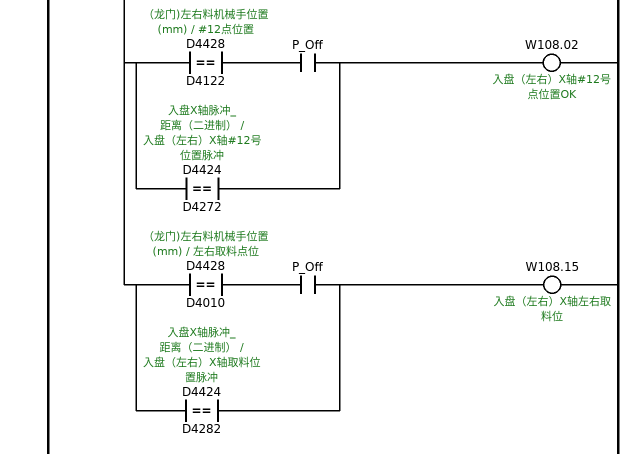
; [picture p264: 入盘机械 / 伺服参数设定, rungs 33-33]
; rung 33: 左右机械手所处位置 / 第一排12点
LD P_On
OUT TR0
LD=SL(303) D4428 D4100  ; （龙门)左右料机械手位置(mm), （龙门）左右#1号点位置
AND P_Off
OR=L(301) D4424 D4250  ; 入盘X轴脉冲_距离（二进制）, 入盘（左右）X轴#1号位置脉冲
ANDLD
OUT W107.07  ; 入盘（左右）X轴#1号点位置ok
LD TR0
LD=SL(303) D4428 D4102  ; （龙门)左右料机械手位置(mm), #2号点位置
AND P_Off
OR=L(301) D4424 D4252  ; 入盘X轴脉冲_距离（二进制）, 入盘（左右）X轴#2号位置脉冲
ANDLD
OUT W107.08  ; 入盘（左右）X轴#2号点位置OK
LD TR0
LD=SL(303) D4428 D4104  ; （龙门)左右料机械手位置(mm), #3点位置
AND P_Off
OR=L(301) D4424 D4254  ; 入盘X轴脉冲_距离（二进制）, 入盘（左右）X轴#3号位置脉冲)
ANDLD
OUT W107.09  ; 入盘（左右）X轴#3号点位置OK
LD TR0
LD=SL(303) D4428 D4106  ; （龙门)左右料机械手位置(mm), #4点位置
AND P_Off
OR=L(301) D4424 D4256  ; 入盘X轴脉冲_距离（二进制）, 入盘（左右）X轴#4号位置脉冲
ANDLD
OUT W107.10  ; 入盘（左右）X轴#4号点位置OK
LD TR0
LD=SL(303) D4428 D4108  ; （龙门)左右料机械手位置(mm), #5点位置
AND P_Off
OR=L(301) D4424 D4258  ; 入盘X轴脉冲_距离（二进制）, 入盘（左右）X轴#5号位置脉冲
ANDLD
OUT W107.11  ; 入盘（左右）X轴#5号点位置OK
LD TR0
LD=SL(303) D4428 D4110  ; （龙门)左右料机械手位置(mm), #6点位置
AND P_Off
OR=L(301) D4424 D4260  ; 入盘X轴脉冲_距离（二进制）, 入盘（左右）X轴#6号位置脉冲
ANDLD
OUT W107.12  ; 入盘（左右）X轴#6号点位置OK
LD TR0
LD=SL(303) D4428 D4112  ; （龙门)左右料机械手位置(mm), #7点位置
AND P_Off
OR=L(301) D4424 D4262  ; 入盘X轴脉冲_距离（二进制）, 入盘（左右）X轴#7号位置脉冲
ANDLD
OUT W107.13  ; 入盘（左右）X轴#7号点位置OK
LD TR0
LD=SL(303) D4428 D4114  ; （龙门)左右料机械手位置(mm), #8点位置
AND P_Off
OR=L(301) D4424 D4264  ; 入盘X轴脉冲_距离（二进制）, 入盘（左右）X轴#8号位置脉冲
ANDLD
OUT W107.14  ; 入盘（左右）X轴#8号点位置OK
LD TR0
LD=SL(303) D4428 D4116  ; （龙门)左右料机械手位置(mm), #9点位置
AND P_Off
OR=L(301) D4424 D4266  ; 入盘X轴脉冲_距离（二进制）, 入盘（左右）X轴#9号位置脉冲
ANDLD
OUT W107.15  ; 入盘（左右）X轴#9号点位置OK
LD TR0
LD=SL(303) D4428 D4118  ; （龙门)左右料机械手位置(mm), #10点位置
AND P_Off
OR=L(301) D4424 D4268  ; 入盘X轴脉冲_距离（二进制）, 入盘（左右）X轴#10号位置脉冲
ANDLD
OUT W108.00  ; 入盘（左右）X轴#10号点位置OK
LD TR0
LD=SL(303) D4428 D4120  ; （龙门)左右料机械手位置(mm), #11点位置
AND P_Off
OR=L(301) D4424 D4270  ; 入盘X轴脉冲_距离（二进制）, 入盘（左右）X轴#11号位置脉冲
ANDLD
OUT W108.01  ; 入盘（左右）X轴#11号点位置OK
LD TR0
LD=SL(303) D4428 D4122  ; （龙门)左右料机械手位置(mm), #12点位置
AND P_Off
OR=L(301) D4424 D4272  ; 入盘X轴脉冲_距离（二进制）, 入盘（左右）X轴#12号位置脉冲
ANDLD
OUT W108.02  ; 入盘（左右）X轴#12号点位置OK
LD TR0
LD=SL(303) D4428 D4010  ; （龙门)左右料机械手位置(mm), 左右取料点位
AND P_Off
OR=L(301) D4424 D4282  ; 入盘X轴脉冲_距离（二进制）, 入盘（左右）X轴取料位置脉冲
ANDLD
OUT W108.15  ; 入盘（左右）X轴左右取料位

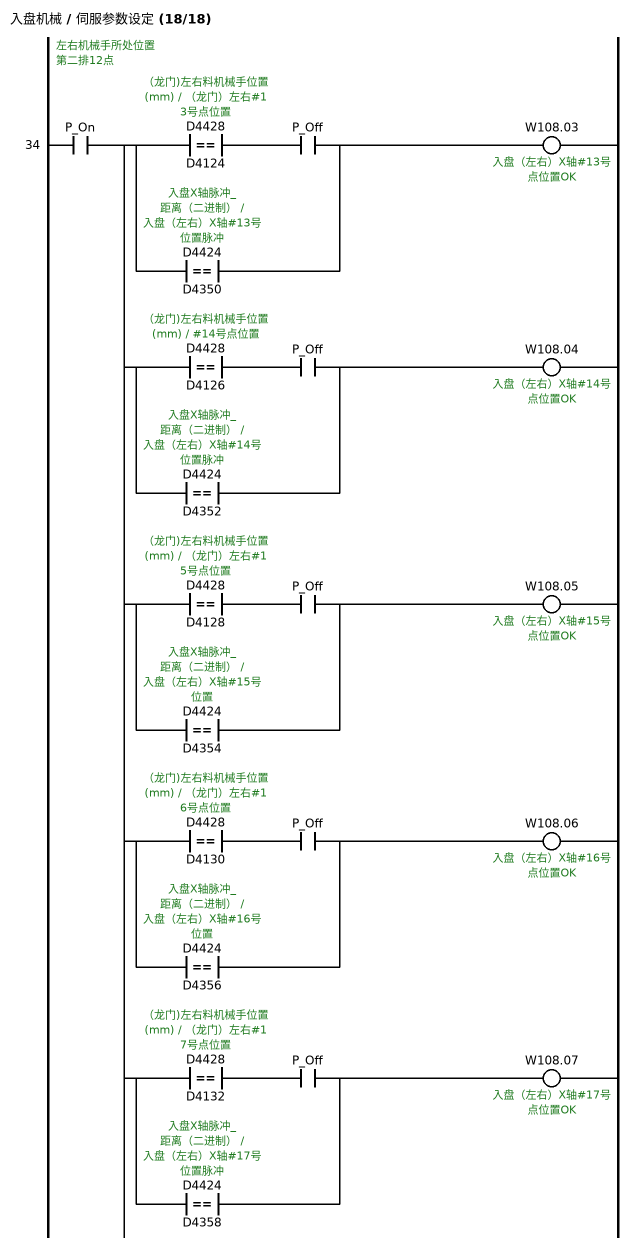

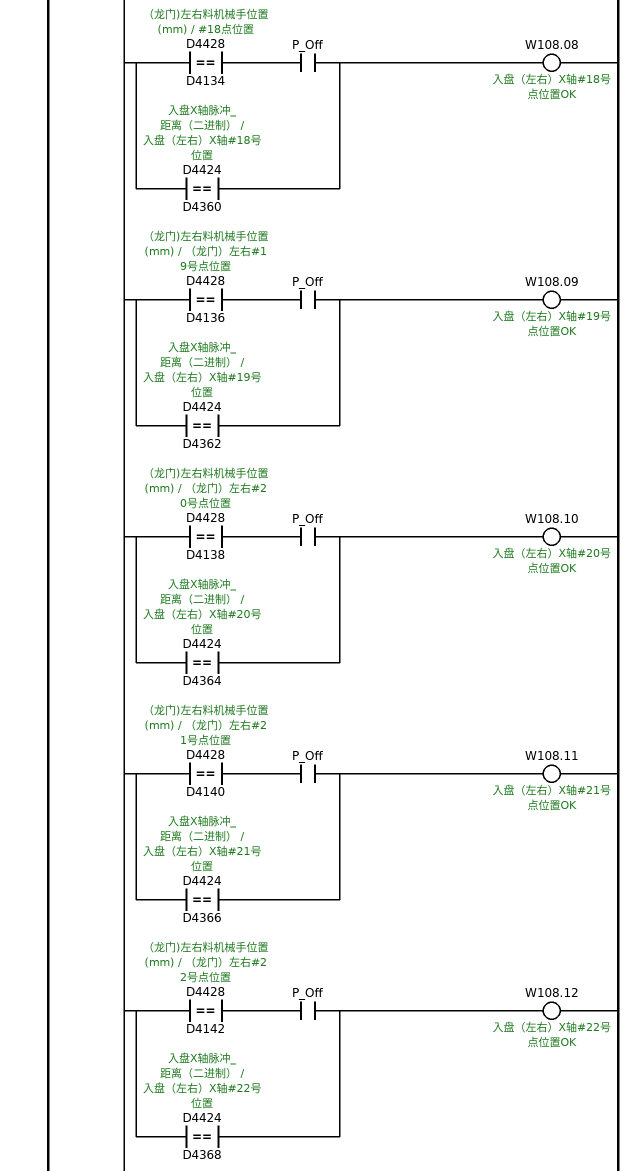

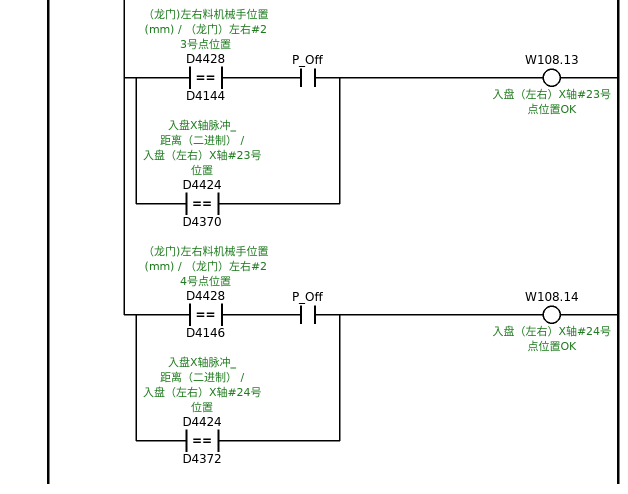
; rung 34: 左右机械手所处位置 / 第二排12点
LD P_On
OUT TR0
LD=SL(303) D4428 D4124  ; （龙门)左右料机械手位置(mm), （龙门）左右#13号点位置
AND P_Off
OR=L(301) D4424 D4350  ; 入盘X轴脉冲_距离（二进制）, 入盘（左右）X轴#13号位置脉冲
ANDLD
OUT W108.03  ; 入盘（左右）X轴#13号点位置OK
LD TR0
LD=SL(303) D4428 D4126  ; （龙门)左右料机械手位置(mm), #14号点位置
AND P_Off
OR=L(301) D4424 D4352  ; 入盘X轴脉冲_距离（二进制）, 入盘（左右）X轴#14号位置脉冲
ANDLD
OUT W108.04  ; 入盘（左右）X轴#14号点位置OK
LD TR0
LD=SL(303) D4428 D4128  ; （龙门)左右料机械手位置(mm), （龙门）左右#15号点位置
AND P_Off
OR=L(301) D4424 D4354  ; 入盘X轴脉冲_距离（二进制）, 入盘（左右）X轴#15号位置
ANDLD
OUT W108.05  ; 入盘（左右）X轴#15号点位置OK
LD TR0
LD=SL(303) D4428 D4130  ; （龙门)左右料机械手位置(mm), （龙门）左右#16号点位置
AND P_Off
OR=L(301) D4424 D4356  ; 入盘X轴脉冲_距离（二进制）, 入盘（左右）X轴#16号位置
ANDLD
OUT W108.06  ; 入盘（左右）X轴#16号点位置OK
LD TR0
LD=SL(303) D4428 D4132  ; （龙门)左右料机械手位置(mm), （龙门）左右#17号点位置
AND P_Off
OR=L(301) D4424 D4358  ; 入盘X轴脉冲_距离（二进制）, 入盘（左右）X轴#17号位置脉冲
ANDLD
OUT W108.07  ; 入盘（左右）X轴#17号点位置OK
LD TR0
LD=SL(303) D4428 D4134  ; （龙门)左右料机械手位置(mm), #18点位置
AND P_Off
OR=L(301) D4424 D4360  ; 入盘X轴脉冲_距离（二进制）, 入盘（左右）X轴#18号位置
ANDLD
OUT W108.08  ; 入盘（左右）X轴#18号点位置OK
LD TR0
LD=SL(303) D4428 D4136  ; （龙门)左右料机械手位置(mm), （龙门）左右#19号点位置
AND P_Off
OR=L(301) D4424 D4362  ; 入盘X轴脉冲_距离（二进制）, 入盘（左右）X轴#19号位置
ANDLD
OUT W108.09  ; 入盘（左右）X轴#19号点位置OK
LD TR0
LD=SL(303) D4428 D4138  ; （龙门)左右料机械手位置(mm), （龙门）左右#20号点位置
AND P_Off
OR=L(301) D4424 D4364  ; 入盘X轴脉冲_距离（二进制）, 入盘（左右）X轴#20号位置
ANDLD
OUT W108.10  ; 入盘（左右）X轴#20号点位置OK
LD TR0
LD=SL(303) D4428 D4140  ; （龙门)左右料机械手位置(mm), （龙门）左右#21号点位置
AND P_Off
OR=L(301) D4424 D4366  ; 入盘X轴脉冲_距离（二进制）, 入盘（左右）X轴#21号位置
ANDLD
OUT W108.11  ; 入盘（左右）X轴#21号点位置OK
LD TR0
LD=SL(303) D4428 D4142  ; （龙门)左右料机械手位置(mm), （龙门）左右#22号点位置
AND P_Off
OR=L(301) D4424 D4368  ; 入盘X轴脉冲_距离（二进制）, 入盘（左右）X轴#22号位置
ANDLD
OUT W108.12  ; 入盘（左右）X轴#22号点位置OK
LD TR0
LD=SL(303) D4428 D4144  ; （龙门)左右料机械手位置(mm), （龙门）左右#23号点位置
AND P_Off
OR=L(301) D4424 D4370  ; 入盘X轴脉冲_距离（二进制）, 入盘（左右）X轴#23号位置
ANDLD
OUT W108.13  ; 入盘（左右）X轴#23号点位置OK
LD TR0
LD=SL(303) D4428 D4146  ; （龙门)左右料机械手位置(mm), （龙门）左右#24号点位置
AND P_Off
OR=L(301) D4424 D4372  ; 入盘X轴脉冲_距离（二进制）, 入盘（左右）X轴#24号位置
ANDLD
OUT W108.14  ; 入盘（左右）X轴#24号点位置OK

### Section 外部输出及轴控运动

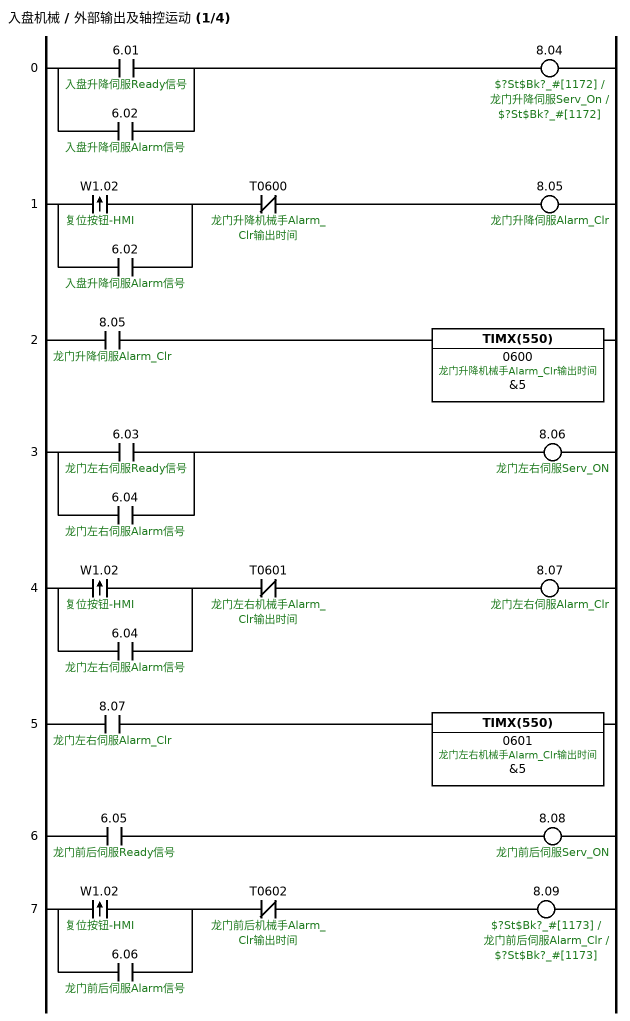
; rung 0
LD 6.01  ; 入盘升降伺服Ready信号
OR 6.02  ; 入盘升降伺服Alarm信号
OUT 8.04  ; $?St$Bk?_#[1172] / 龙门升降伺服Serv_On / $?St$Bk?_#[1172]
; rung 1
@LD W1.02  ; 复位按钮-HMI
OR 6.02  ; 入盘升降伺服Alarm信号
ANDNOT T0600  ; 龙门升降机械手Alarm_Clr输出时间
OUT 8.05  ; 龙门升降伺服Alarm_Clr
; rung 2
LD 8.05  ; 龙门升降伺服Alarm_Clr
TIMX(550) 0600 &5  ; 龙门升降机械手Alarm_Clr输出时间
; rung 3
LD 6.03  ; 龙门左右伺服Ready信号
OR 6.04  ; 龙门左右伺服Alarm信号
OUT 8.06  ; 龙门左右伺服Serv_ON
; rung 4
@LD W1.02  ; 复位按钮-HMI
OR 6.04  ; 龙门左右伺服Alarm信号
ANDNOT T0601  ; 龙门左右机械手Alarm_Clr输出时间
OUT 8.07  ; 龙门左右伺服Alarm_Clr
; rung 5
LD 8.07  ; 龙门左右伺服Alarm_Clr
TIMX(550) 0601 &5  ; 龙门左右机械手Alarm_Clr输出时间
; rung 6
LD 6.05  ; 龙门前后伺服Ready信号
OUT 8.08  ; 龙门前后伺服Serv_ON
; rung 7
@LD W1.02  ; 复位按钮-HMI
OR 6.06  ; 龙门前后伺服Alarm信号
ANDNOT T0602  ; 龙门前后机械手Alarm_Clr输出时间
OUT 8.09  ; $?St$Bk?_#[1173] / 龙门前后伺服Alarm_Clr / $?St$Bk?_#[1173]

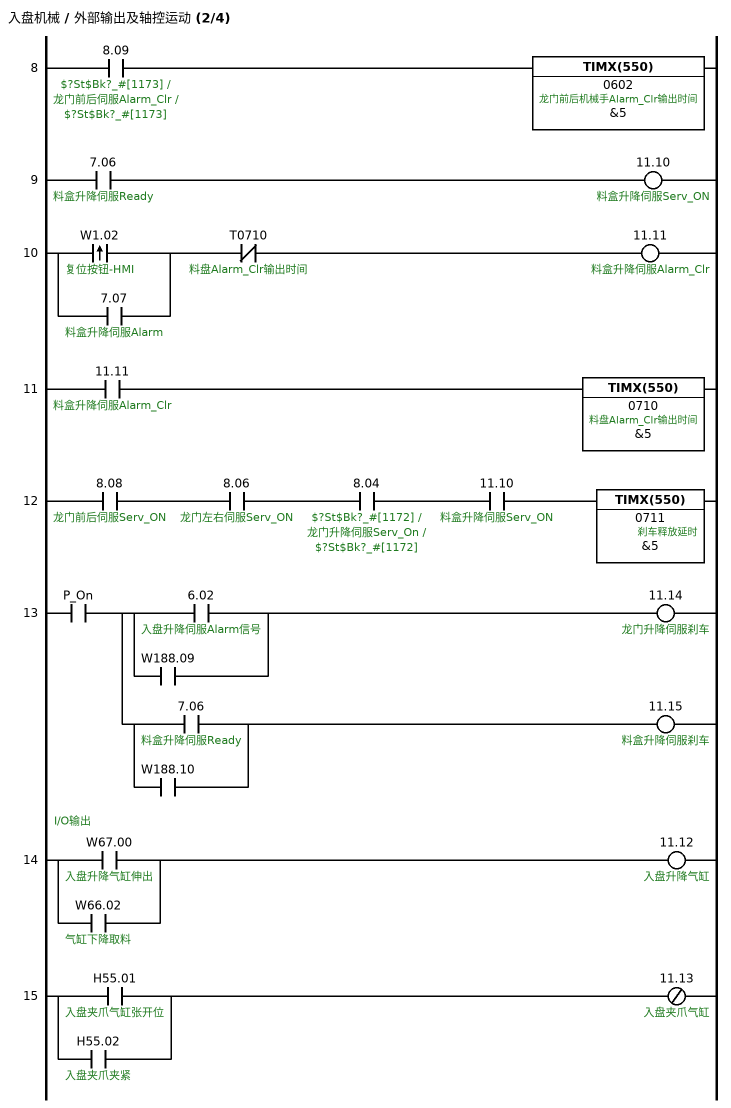
; rung 8
LD 8.09  ; $?St$Bk?_#[1173] / 龙门前后伺服Alarm_Clr / $?St$Bk?_#[1173]
TIMX(550) 0602 &5  ; 龙门前后机械手Alarm_Clr输出时间
; rung 9
LD 7.06  ; 料盒升降伺服Ready
OUT 11.10  ; 料盒升降伺服Serv_ON
; rung 10
@LD W1.02  ; 复位按钮-HMI
OR 7.07  ; 料盒升降伺服Alarm
ANDNOT T0710  ; 料盘Alarm_Clr输出时间
OUT 11.11  ; 料盒升降伺服Alarm_Clr
; rung 11
LD 11.11  ; 料盒升降伺服Alarm_Clr
TIMX(550) 0710 &5  ; 料盘Alarm_Clr输出时间
; rung 12
LD 8.08  ; 龙门前后伺服Serv_ON
AND 8.06  ; 龙门左右伺服Serv_ON
AND 8.04  ; $?St$Bk?_#[1172] / 龙门升降伺服Serv_On / $?St$Bk?_#[1172]
AND 11.10  ; 料盒升降伺服Serv_ON
TIMX(550) 0711 &5  ; 刹车释放延时
; rung 13
LD P_On
OUT TR0
LD 6.02  ; 入盘升降伺服Alarm信号
OR W188.09
ANDLD
OUT 11.14  ; 龙门升降伺服刹车
LD TR0
LD 7.06  ; 料盒升降伺服Ready
OR W188.10
ANDLD
OUT 11.15  ; 料盒升降伺服刹车
; rung 14: I/O输出
LD W67.00  ; 入盘升降气缸伸出
OR W66.02  ; 气缸下降取料
OUT 11.12  ; 入盘升降气缸
; rung 15
LD H55.01  ; 入盘夹爪气缸张开位
OR H55.02  ; 入盘夹爪夹紧
OUTNOT 11.13  ; 入盘夹爪气缸

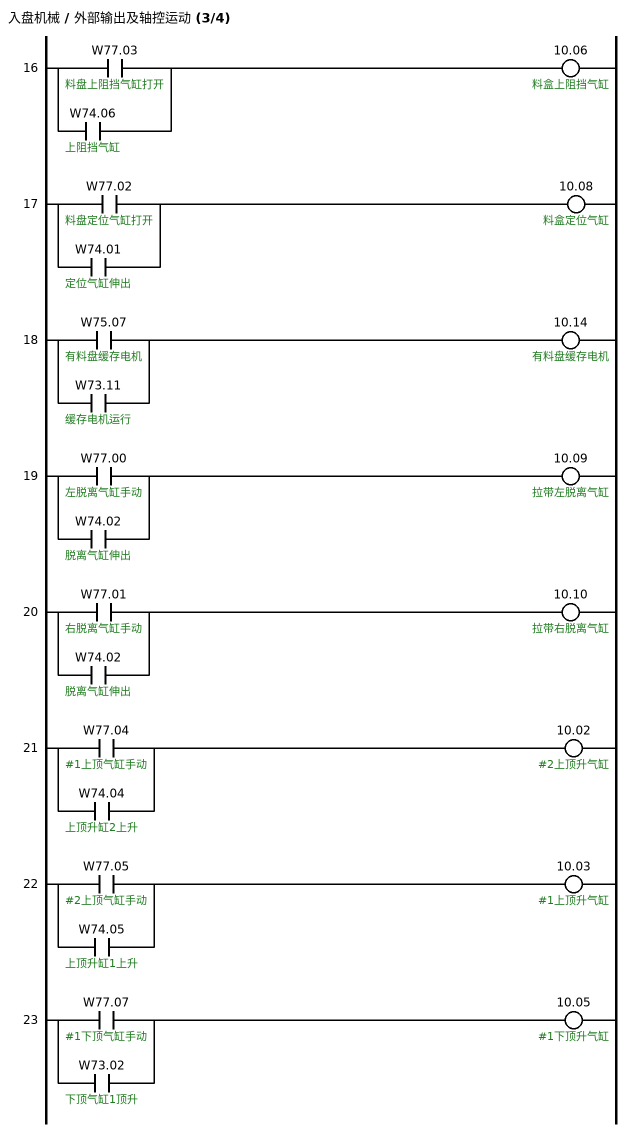
; rung 16
LD W77.03  ; 料盘上阻挡气缸打开
OR W74.06  ; 上阻挡气缸
OUT 10.06  ; 料盒上阻挡气缸
; rung 17
LD W77.02  ; 料盘定位气缸打开
OR W74.01  ; 定位气缸伸出
OUT 10.08  ; 料盒定位气缸
; rung 18
LD W75.07  ; 有料盘缓存电机
OR W73.11  ; 缓存电机运行
OUT 10.14  ; 有料盘缓存电机
; rung 19
LD W77.00  ; 左脱离气缸手动
OR W74.02  ; 脱离气缸伸出
OUT 10.09  ; 拉带左脱离气缸
; rung 20
LD W77.01  ; 右脱离气缸手动
OR W74.02  ; 脱离气缸伸出
OUT 10.10  ; 拉带右脱离气缸
; rung 21
LD W77.04  ; #1上顶气缸手动
OR W74.04  ; 上顶升缸2上升
OUT 10.02  ; #2上顶升气缸
; rung 22
LD W77.05  ; #2上顶气缸手动
OR W74.05  ; 上顶升缸1上升
OUT 10.03  ; #1上顶升气缸
; rung 23
LD W77.07  ; #1下顶气缸手动
OR W73.02  ; 下顶气缸1顶升
OUT 10.05  ; #1下顶升气缸

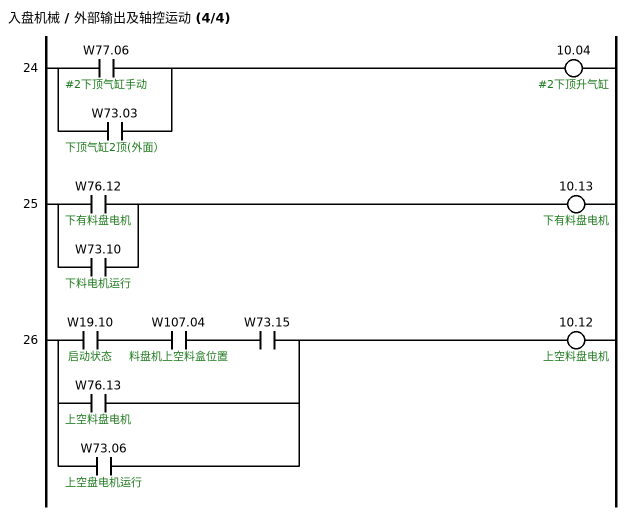
; rung 24
LD W77.06  ; #2下顶气缸手动
OR W73.03  ; 下顶气缸2顶(外面）
OUT 10.04  ; #2下顶升气缸
; rung 25
LD W76.12  ; 下有料盘电机
OR W73.10  ; 下料电机运行
OUT 10.13  ; 下有料盘电机
; rung 26
LD W19.10  ; 启动状态
AND W107.04  ; 料盘机上空料盒位置
AND W73.15
OR W76.13  ; 上空料盘电机
OR W73.06  ; 上空盘电机运行
OUT 10.12  ; 上空料盘电机

### Section 自动报警

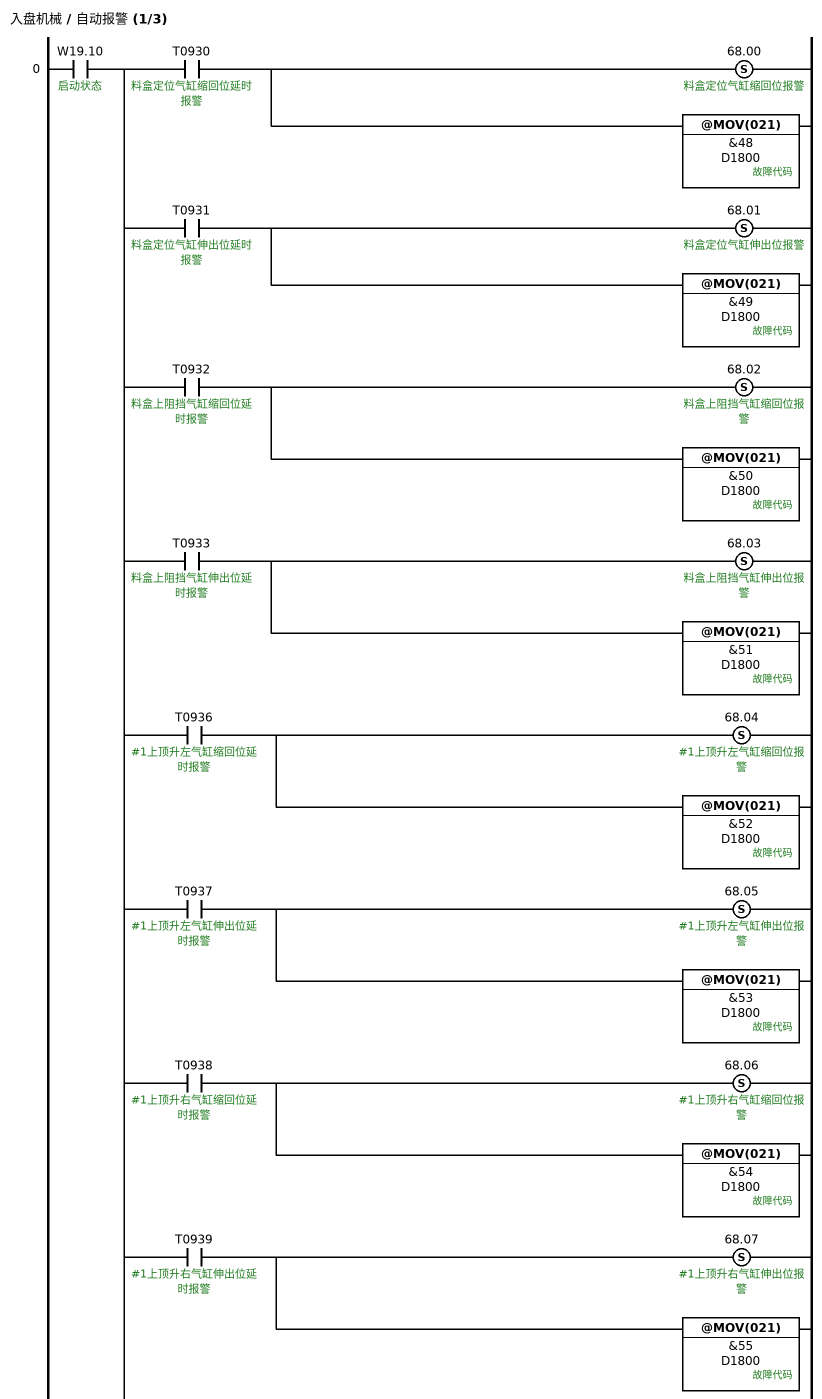

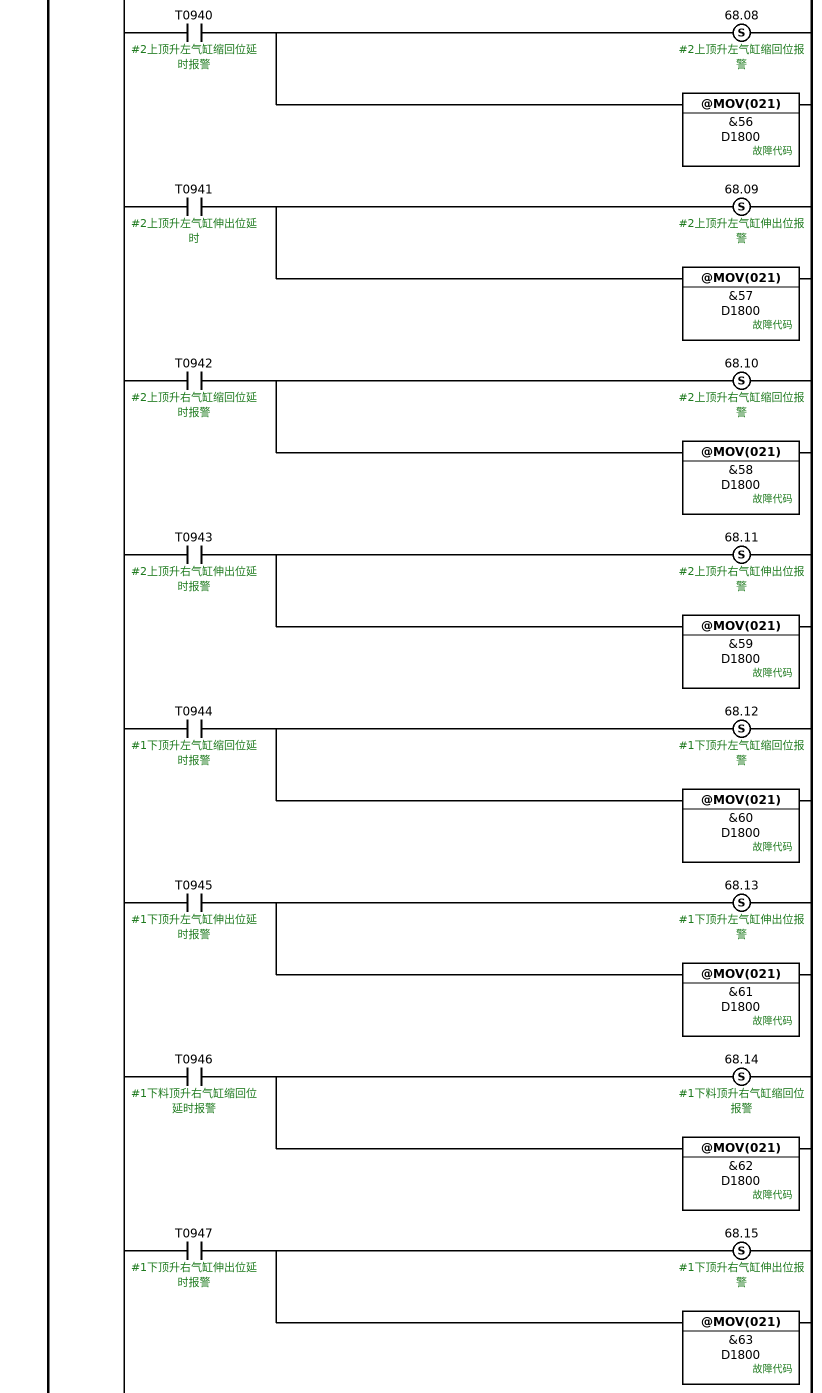

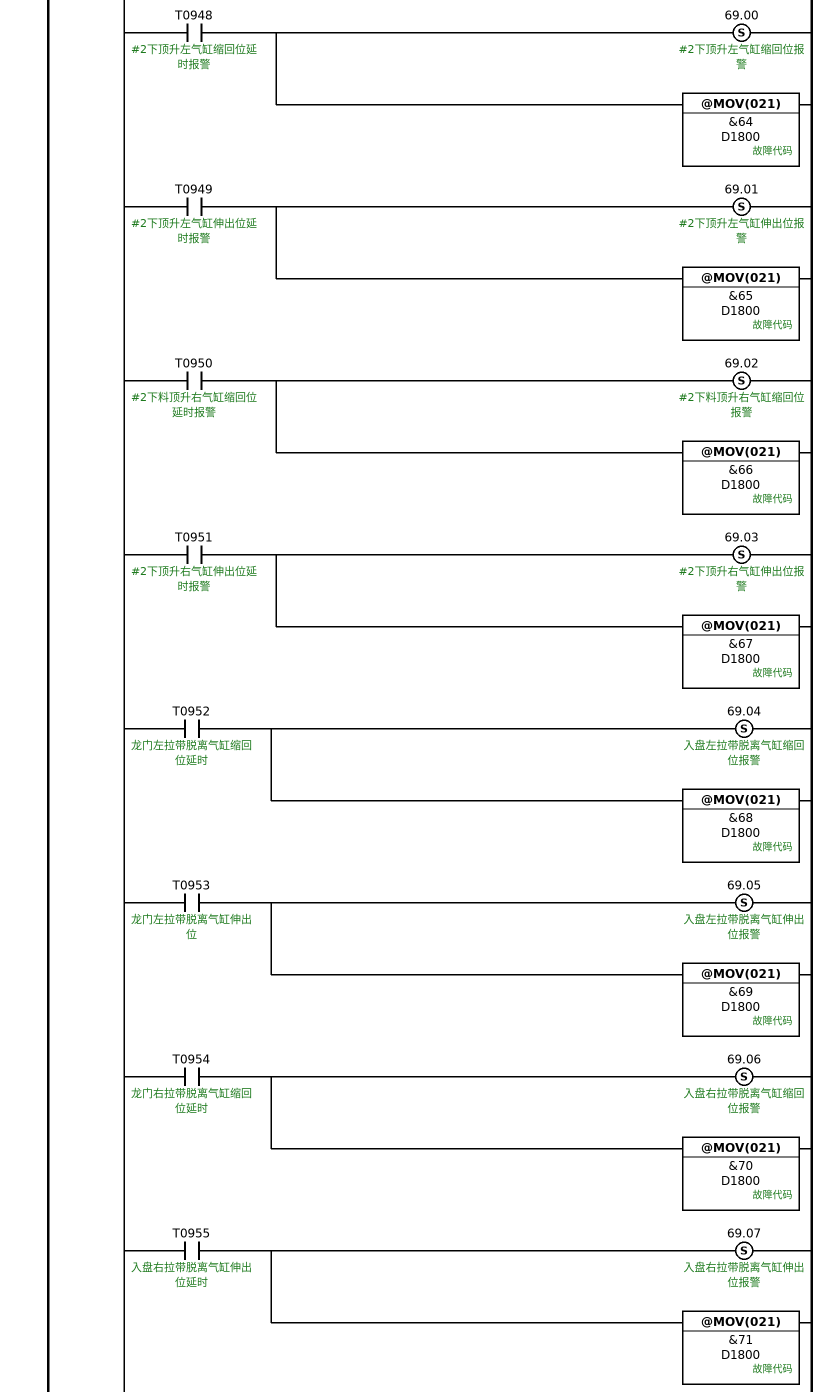

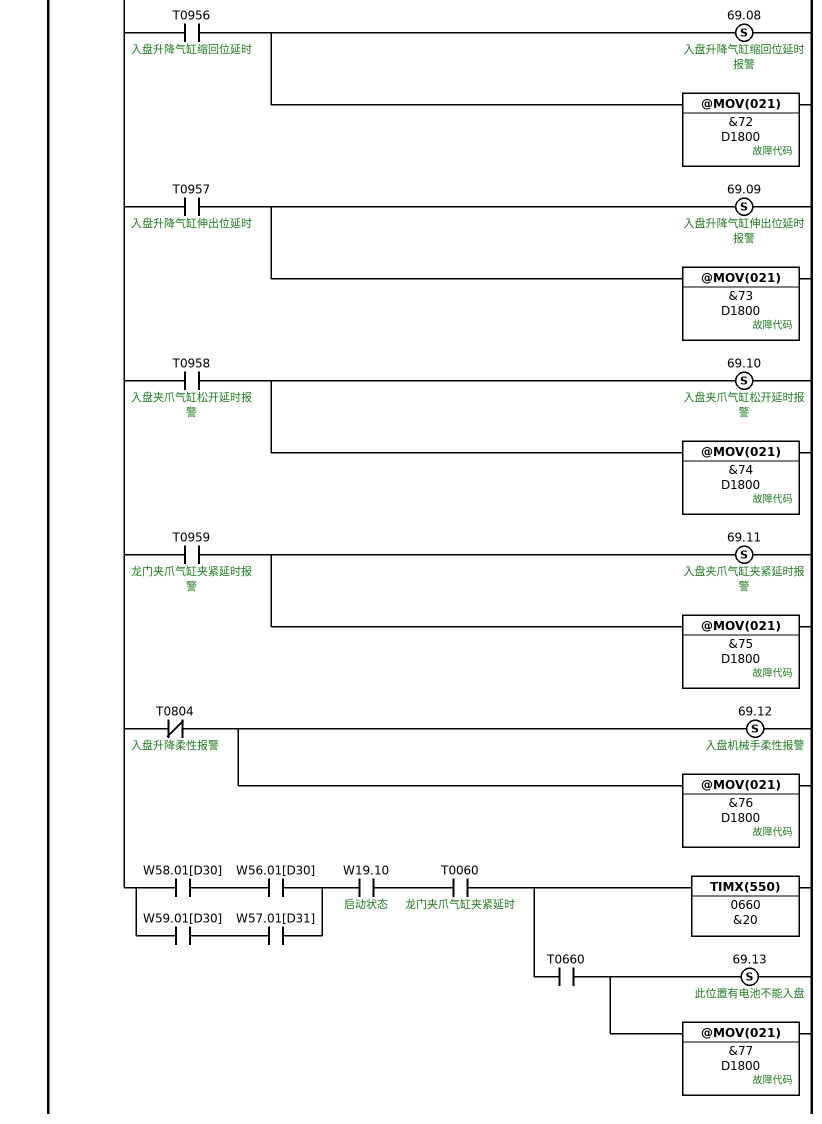
; rung 0
LD W19.10  ; 启动状态
OUT TR0
AND T0930  ; 料盒定位气缸缩回位延时报警
SET 68.00  ; 料盒定位气缸缩回位报警
@MOV(021) &48 D1800  ; 故障代码
LD TR0
AND T0931  ; 料盒定位气缸伸出位延时报警
SET 68.01  ; 料盒定位气缸伸出位报警
@MOV(021) &49 D1800  ; 故障代码
LD TR0
AND T0932  ; 料盒上阻挡气缸缩回位延时报警
SET 68.02  ; 料盒上阻挡气缸缩回位报警
@MOV(021) &50 D1800  ; 故障代码
LD TR0
AND T0933  ; 料盒上阻挡气缸伸出位延时报警
SET 68.03  ; 料盒上阻挡气缸伸出位报警
@MOV(021) &51 D1800  ; 故障代码
LD TR0
AND T0936  ; #1上顶升左气缸缩回位延时报警
SET 68.04  ; #1上顶升左气缸缩回位报警
@MOV(021) &52 D1800  ; 故障代码
LD TR0
AND T0937  ; #1上顶升左气缸伸出位延时报警
SET 68.05  ; #1上顶升左气缸伸出位报警
@MOV(021) &53 D1800  ; 故障代码
LD TR0
AND T0938  ; #1上顶升右气缸缩回位延时报警
SET 68.06  ; #1上顶升右气缸缩回位报警
@MOV(021) &54 D1800  ; 故障代码
LD TR0
AND T0939  ; #1上顶升右气缸伸出位延时报警
SET 68.07  ; #1上顶升右气缸伸出位报警
@MOV(021) &55 D1800  ; 故障代码
LD TR0
AND T0940  ; #2上顶升左气缸缩回位延时报警
SET 68.08  ; #2上顶升左气缸缩回位报警
@MOV(021) &56 D1800  ; 故障代码
LD TR0
AND T0941  ; #2上顶升左气缸伸出位延时
SET 68.09  ; #2上顶升左气缸伸出位报警
@MOV(021) &57 D1800  ; 故障代码
LD TR0
AND T0942  ; #2上顶升右气缸缩回位延时报警
SET 68.10  ; #2上顶升右气缸缩回位报警
@MOV(021) &58 D1800  ; 故障代码
LD TR0
AND T0943  ; #2上顶升右气缸伸出位延时报警
SET 68.11  ; #2上顶升右气缸伸出位报警
@MOV(021) &59 D1800  ; 故障代码
LD TR0
AND T0944  ; #1下顶升左气缸缩回位延时报警
SET 68.12  ; #1下顶升左气缸缩回位报警
@MOV(021) &60 D1800  ; 故障代码
LD TR0
AND T0945  ; #1下顶升左气缸伸出位延时报警
SET 68.13  ; #1下顶升左气缸伸出位报警
@MOV(021) &61 D1800  ; 故障代码
LD TR0
AND T0946  ; #1下料顶升右气缸缩回位延时报警
SET 68.14  ; #1下料顶升右气缸缩回位报警
@MOV(021) &62 D1800  ; 故障代码
LD TR0
AND T0947  ; #1下顶升右气缸伸出位延时报警
SET 68.15  ; #1下顶升右气缸伸出位报警
@MOV(021) &63 D1800  ; 故障代码
LD TR0
AND T0948  ; #2下顶升左气缸缩回位延时报警
SET 69.00  ; #2下顶升左气缸缩回位报警
@MOV(021) &64 D1800  ; 故障代码
LD TR0
AND T0949  ; #2下顶升左气缸伸出位延时报警
SET 69.01  ; #2下顶升左气缸伸出位报警
@MOV(021) &65 D1800  ; 故障代码
LD TR0
AND T0950  ; #2下料顶升右气缸缩回位延时报警
SET 69.02  ; #2下料顶升右气缸缩回位报警
@MOV(021) &66 D1800  ; 故障代码
LD TR0
AND T0951  ; #2下顶升右气缸伸出位延时报警
SET 69.03  ; #2下顶升右气缸伸出位报警
@MOV(021) &67 D1800  ; 故障代码
LD TR0
AND T0952  ; 龙门左拉带脱离气缸缩回位延时
SET 69.04  ; 入盘左拉带脱离气缸缩回位报警
@MOV(021) &68 D1800  ; 故障代码
LD TR0
AND T0953  ; 龙门左拉带脱离气缸伸出位
SET 69.05  ; 入盘左拉带脱离气缸伸出位报警
@MOV(021) &69 D1800  ; 故障代码
LD TR0
AND T0954  ; 龙门右拉带脱离气缸缩回位延时
SET 69.06  ; 入盘右拉带脱离气缸缩回位报警
@MOV(021) &70 D1800  ; 故障代码
LD TR0
AND T0955  ; 入盘右拉带脱离气缸伸出位延时
SET 69.07  ; 入盘右拉带脱离气缸伸出位报警
@MOV(021) &71 D1800  ; 故障代码
LD TR0
AND T0956  ; 入盘升降气缸缩回位延时
SET 69.08  ; 入盘升降气缸缩回位延时报警
@MOV(021) &72 D1800  ; 故障代码
LD TR0
AND T0957  ; 入盘升降气缸伸出位延时
SET 69.09  ; 入盘升降气缸伸出位延时报警
@MOV(021) &73 D1800  ; 故障代码
LD TR0
AND T0958  ; 入盘夹爪气缸松开延时报警
SET 69.10  ; 入盘夹爪气缸松开延时报警
@MOV(021) &74 D1800  ; 故障代码
LD TR0
AND T0959  ; 龙门夹爪气缸夹紧延时报警
SET 69.11  ; 入盘夹爪气缸夹紧延时报警
@MOV(021) &75 D1800  ; 故障代码
LD TR0
ANDNOT T0804  ; 入盘升降柔性报警
SET 69.12  ; 入盘机械手柔性报警
@MOV(021) &76 D1800  ; 故障代码
LD TR0
LD W58.01[D30]
AND W56.01[D30]
LD W59.01[D30]
AND W57.01[D31]
ORLD
ANDLD
AND W19.10  ; 启动状态
AND T0060  ; 龙门夹爪气缸夹紧延时
TIMX(550) 0660 &20
AND T0660
SET 69.13  ; 此位置有电池不能入盘
@MOV(021) &77 D1800  ; 故障代码

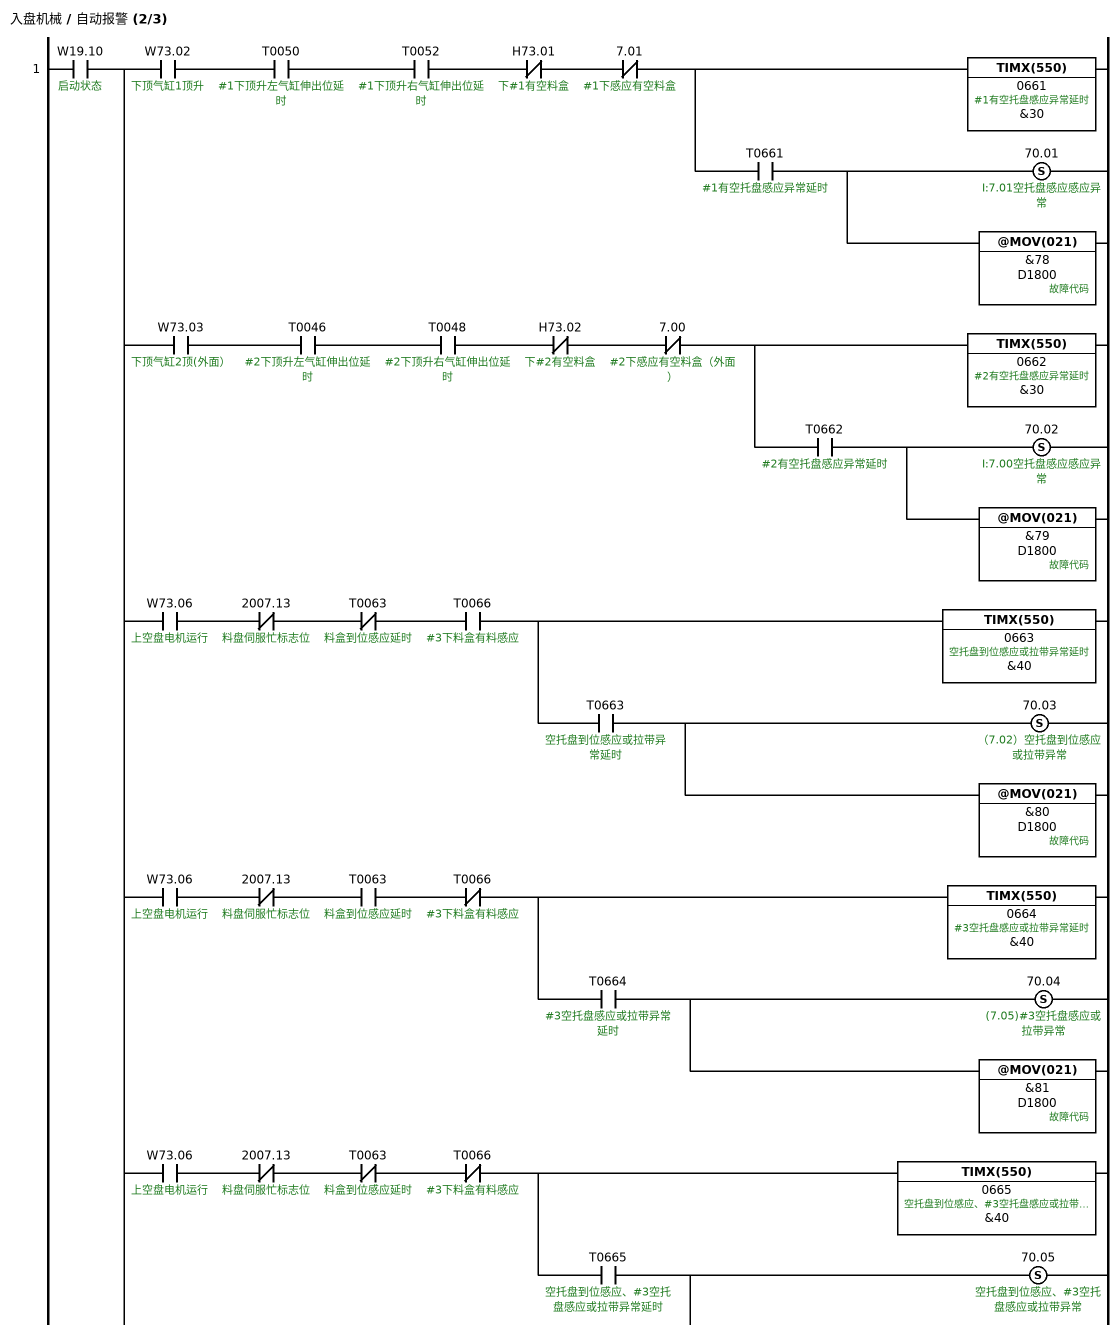

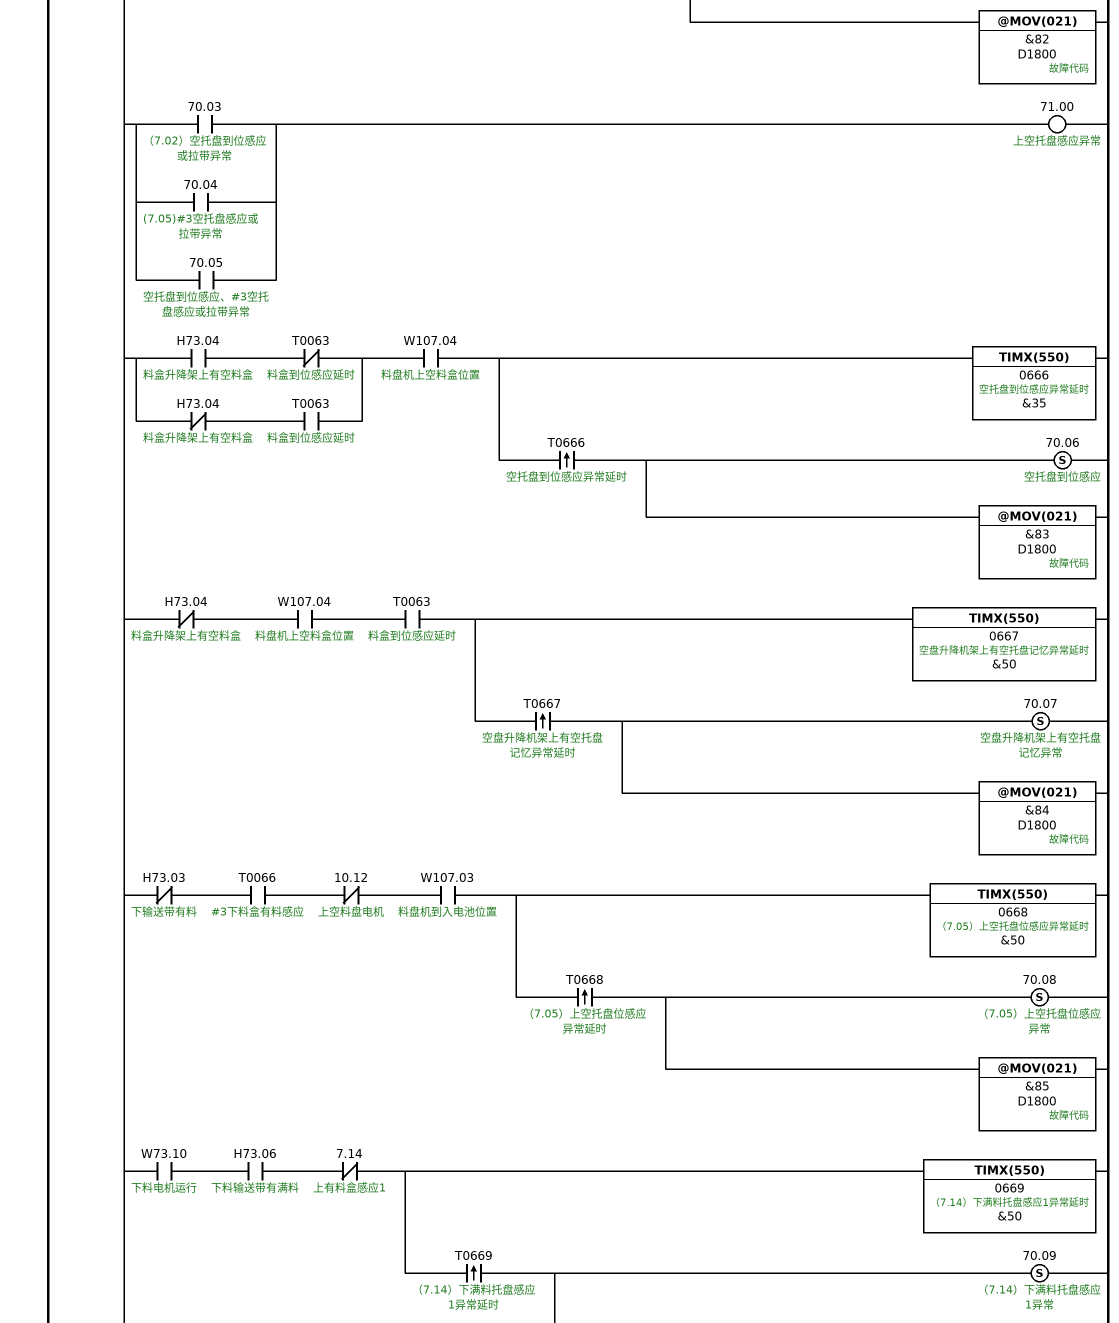

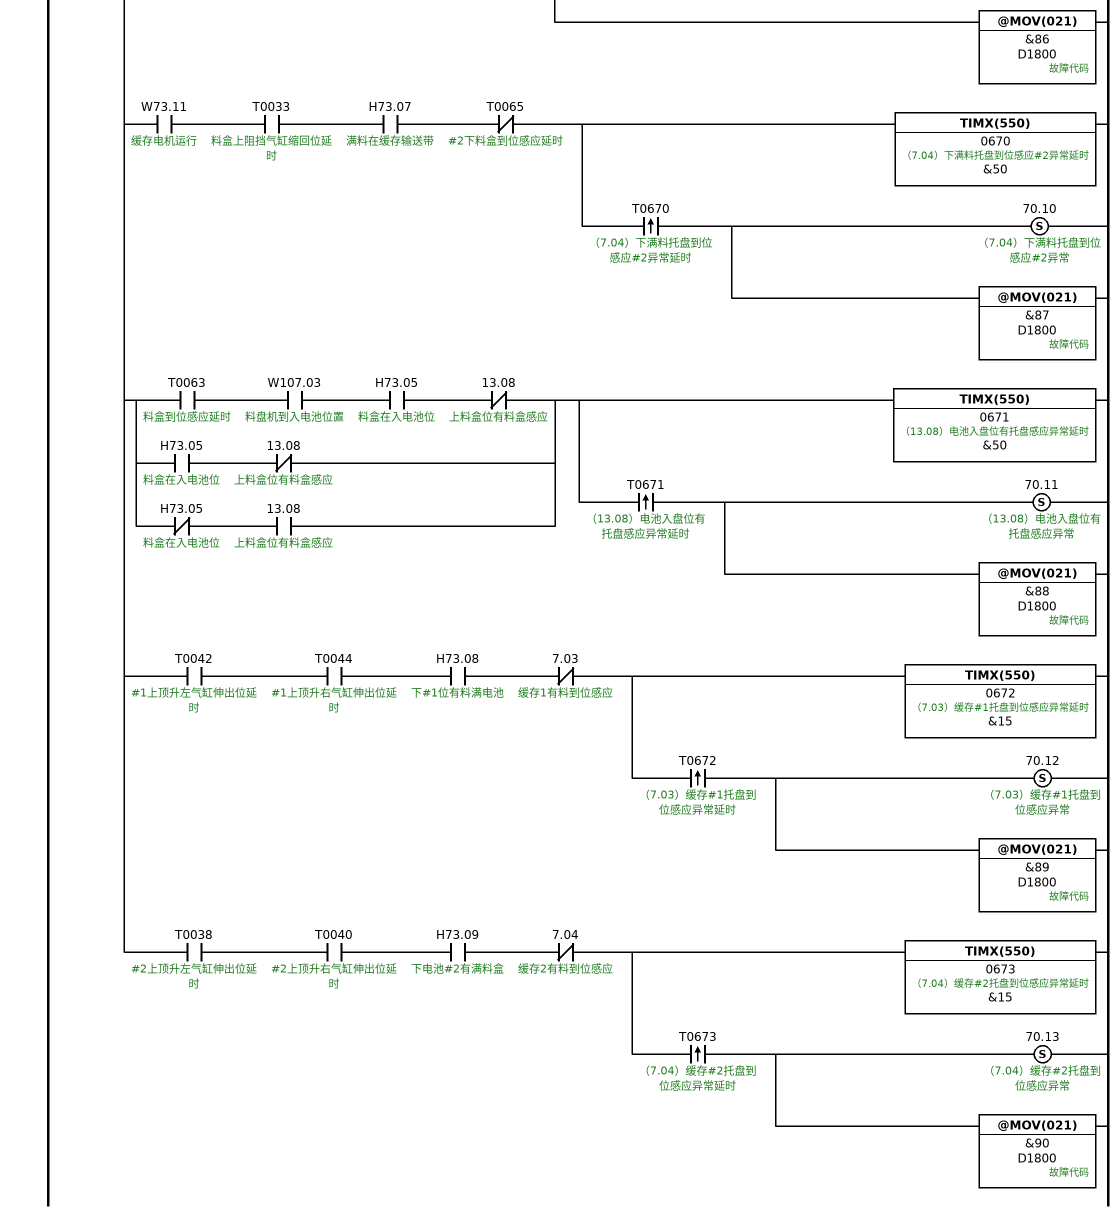
; rung 1
LD W19.10  ; 启动状态
OUT TR0
AND W73.02  ; 下顶气缸1顶升
AND T0050  ; #1下顶升左气缸伸出位延时
AND T0052  ; #1下顶升右气缸伸出位延时
ANDNOT H73.01  ; 下#1有空料盒
ANDNOT 7.01  ; #1下感应有空料盒
TIMX(550) 0661 &30  ; #1有空托盘感应异常延时
AND T0661  ; #1有空托盘感应异常延时
SET 70.01  ; I:7.01空托盘感应感应异常
@MOV(021) &78 D1800  ; 故障代码
LD TR0
AND W73.03  ; 下顶气缸2顶(外面）
AND T0046  ; #2下顶升左气缸伸出位延时
AND T0048  ; #2下顶升右气缸伸出位延时
ANDNOT H73.02  ; 下#2有空料盒
ANDNOT 7.00  ; #2下感应有空料盒（外面）
TIMX(550) 0662 &30  ; #2有空托盘感应异常延时
AND T0662  ; #2有空托盘感应异常延时
SET 70.02  ; I:7.00空托盘感应感应异常
@MOV(021) &79 D1800  ; 故障代码
LD TR0
AND W73.06  ; 上空盘电机运行
ANDNOT 2007.13  ; 料盘伺服忙标志位
ANDNOT T0063  ; 料盒到位感应延时
AND T0066  ; #3下料盒有料感应
TIMX(550) 0663 &40  ; 空托盘到位感应或拉带异常延时
AND T0663  ; 空托盘到位感应或拉带异常延时
SET 70.03  ; （7.02）空托盘到位感应或拉带异常
@MOV(021) &80 D1800  ; 故障代码
LD TR0
AND W73.06  ; 上空盘电机运行
ANDNOT 2007.13  ; 料盘伺服忙标志位
AND T0063  ; 料盒到位感应延时
ANDNOT T0066  ; #3下料盒有料感应
TIMX(550) 0664 &40  ; #3空托盘感应或拉带异常延时
AND T0664  ; #3空托盘感应或拉带异常延时
SET 70.04  ; (7.05)#3空托盘感应或拉带异常
@MOV(021) &81 D1800  ; 故障代码
LD TR0
AND W73.06  ; 上空盘电机运行
ANDNOT 2007.13  ; 料盘伺服忙标志位
ANDNOT T0063  ; 料盒到位感应延时
ANDNOT T0066  ; #3下料盒有料感应
TIMX(550) 0665 &40  ; 空托盘到位感应、#3空托盘感应或拉带异常延时
AND T0665  ; 空托盘到位感应、#3空托盘感应或拉带异常延时
SET 70.05  ; 空托盘到位感应、#3空托盘感应或拉带异常
@MOV(021) &82 D1800  ; 故障代码
LD TR0
LD 70.03  ; （7.02）空托盘到位感应或拉带异常
OR 70.04  ; (7.05)#3空托盘感应或拉带异常
OR 70.05  ; 空托盘到位感应、#3空托盘感应或拉带异常
ANDLD
OUT 71.00  ; 上空托盘感应异常
LD TR0
LD H73.04  ; 料盒升降架上有空料盒
ANDNOT T0063  ; 料盒到位感应延时
LDNOT H73.04  ; 料盒升降架上有空料盒
AND T0063  ; 料盒到位感应延时
ORLD
ANDLD
AND W107.04  ; 料盘机上空料盒位置
TIMX(550) 0666 &35  ; 空托盘到位感应异常延时
@AND T0666  ; 空托盘到位感应异常延时
SET 70.06  ; 空托盘到位感应
@MOV(021) &83 D1800  ; 故障代码
LD TR0
ANDNOT H73.04  ; 料盒升降架上有空料盒
AND W107.04  ; 料盘机上空料盒位置
AND T0063  ; 料盒到位感应延时
TIMX(550) 0667 &50  ; 空盘升降机架上有空托盘记忆异常延时
@AND T0667  ; 空盘升降机架上有空托盘记忆异常延时
SET 70.07  ; 空盘升降机架上有空托盘记忆异常
@MOV(021) &84 D1800  ; 故障代码
LD TR0
ANDNOT H73.03  ; 下输送带有料
AND T0066  ; #3下料盒有料感应
ANDNOT 10.12  ; 上空料盘电机
AND W107.03  ; 料盘机到入电池位置
TIMX(550) 0668 &50  ; （7.05）上空托盘位感应异常延时
@AND T0668  ; （7.05）上空托盘位感应异常延时
SET 70.08  ; （7.05）上空托盘位感应异常
@MOV(021) &85 D1800  ; 故障代码
LD TR0
AND W73.10  ; 下料电机运行
AND H73.06  ; 下料输送带有满料
ANDNOT 7.14  ; 上有料盒感应1
TIMX(550) 0669 &50  ; （7.14）下满料托盘感应1异常延时
@AND T0669  ; （7.14）下满料托盘感应1异常延时
SET 70.09  ; （7.14）下满料托盘感应1异常
@MOV(021) &86 D1800  ; 故障代码
LD TR0
AND W73.11  ; 缓存电机运行
AND T0033  ; 料盒上阻挡气缸缩回位延时
AND H73.07  ; 满料在缓存输送带
ANDNOT T0065  ; #2下料盒到位感应延时
TIMX(550) 0670 &50  ; （7.04）下满料托盘到位感应#2异常延时
@AND T0670  ; （7.04）下满料托盘到位感应#2异常延时
SET 70.10  ; （7.04）下满料托盘到位感应#2异常
@MOV(021) &87 D1800  ; 故障代码
LD TR0
LD T0063  ; 料盒到位感应延时
AND W107.03  ; 料盘机到入电池位置
AND H73.05  ; 料盒在入电池位
ANDNOT 13.08  ; 上料盒位有料盒感应
LD H73.05  ; 料盒在入电池位
ANDNOT 13.08  ; 上料盒位有料盒感应
ORLD
LDNOT H73.05  ; 料盒在入电池位
AND 13.08  ; 上料盒位有料盒感应
ORLD
ANDLD
TIMX(550) 0671 &50  ; （13.08）电池入盘位有托盘感应异常延时
@AND T0671  ; （13.08）电池入盘位有托盘感应异常延时
SET 70.11  ; （13.08）电池入盘位有托盘感应异常
@MOV(021) &88 D1800  ; 故障代码
LD TR0
AND T0042  ; #1上顶升左气缸伸出位延时
AND T0044  ; #1上顶升右气缸伸出位延时
AND H73.08  ; 下#1位有料满电池
ANDNOT 7.03  ; 缓存1有料到位感应
TIMX(550) 0672 &15  ; （7.03）缓存#1托盘到位感应异常延时
@AND T0672  ; （7.03）缓存#1托盘到位感应异常延时
SET 70.12  ; （7.03）缓存#1托盘到位感应异常
@MOV(021) &89 D1800  ; 故障代码
LD TR0
AND T0038  ; #2上顶升左气缸伸出位延时
AND T0040  ; #2上顶升右气缸伸出位延时
AND H73.09  ; 下电池#2有满料盒
ANDNOT 7.04  ; 缓存2有料到位感应
TIMX(550) 0673 &15  ; （7.04）缓存#2托盘到位感应异常延时
@AND T0673  ; （7.04）缓存#2托盘到位感应异常延时
SET 70.13  ; （7.04）缓存#2托盘到位感应异常
@MOV(021) &90 D1800  ; 故障代码

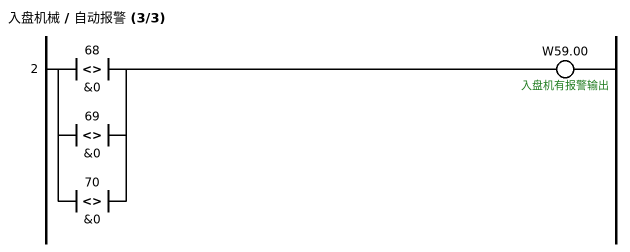
; rung 2
LD<>(305) 68 &0
OR<>(305) 69 &0
OR<>(305) 70 &0
OUT W59.00  ; 入盘机有报警输出

### Section 入盘机构复位

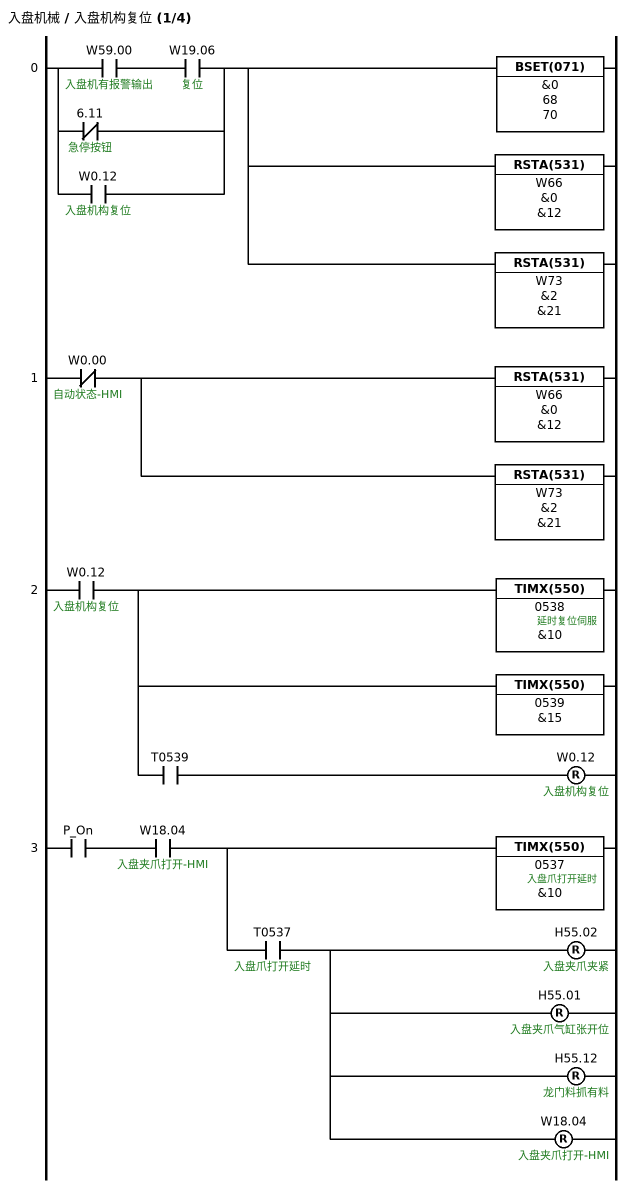
; rung 0
LD W59.00  ; 入盘机有报警输出
AND W19.06  ; 复位
ORNOT 6.11  ; 急停按钮
OR W0.12  ; 入盘机构复位
BSET(071) &0 68 70
RSTA(531) W66 &0 &12
RSTA(531) W73 &2 &21
; rung 1
LDNOT W0.00  ; 自动状态-HMI
RSTA(531) W66 &0 &12
RSTA(531) W73 &2 &21
; rung 2
LD W0.12  ; 入盘机构复位
TIMX(550) 0538 &10  ; 延时复位伺服
TIMX(550) 0539 &15
AND T0539
RSET W0.12  ; 入盘机构复位
; rung 3
LD P_On
AND W18.04  ; 入盘夹爪打开-HMI
TIMX(550) 0537 &10  ; 入盘爪打开延时
AND T0537  ; 入盘爪打开延时
RSET H55.02  ; 入盘夹爪夹紧
RSET H55.01  ; 入盘夹爪气缸张开位
RSET H55.12  ; 龙门料抓有料
RSET W18.04  ; 入盘夹爪打开-HMI

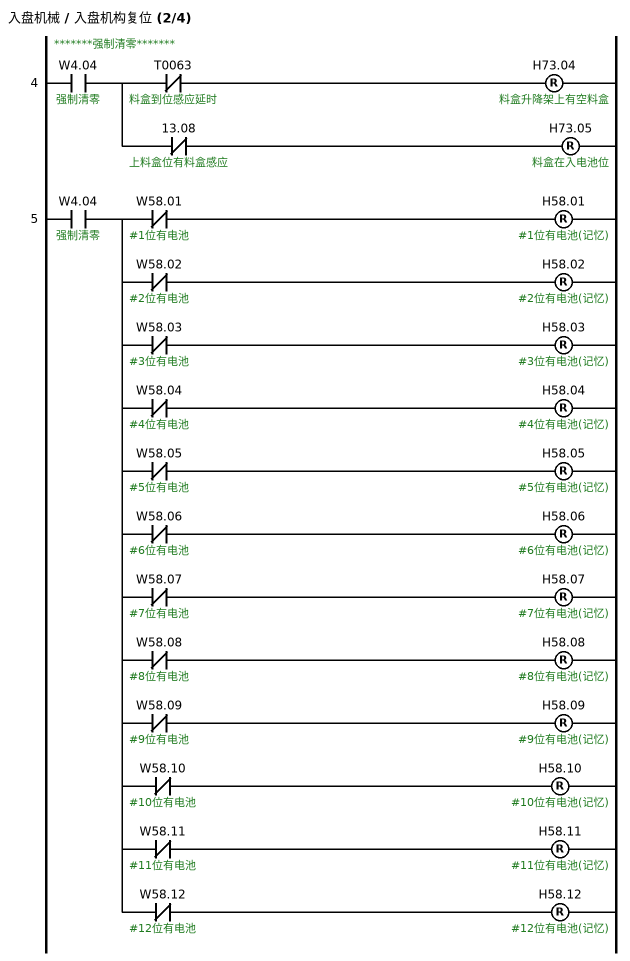
; rung 4: *******强制清零*******
LD W4.04  ; 强制清零
OUT TR0
ANDNOT T0063  ; 料盒到位感应延时
RSET H73.04  ; 料盒升降架上有空料盒
LD TR0
ANDNOT 13.08  ; 上料盒位有料盒感应
RSET H73.05  ; 料盒在入电池位
; rung 5
LD W4.04  ; 强制清零
OUT TR0
ANDNOT W58.01  ; #1位有电池
RSET H58.01  ; #1位有电池(记忆)
LD TR0
ANDNOT W58.02  ; #2位有电池
RSET H58.02  ; #2位有电池(记忆)
LD TR0
ANDNOT W58.03  ; #3位有电池
RSET H58.03  ; #3位有电池(记忆)
LD TR0
ANDNOT W58.04  ; #4位有电池
RSET H58.04  ; #4位有电池(记忆)
LD TR0
ANDNOT W58.05  ; #5位有电池
RSET H58.05  ; #5位有电池(记忆)
LD TR0
ANDNOT W58.06  ; #6位有电池
RSET H58.06  ; #6位有电池(记忆)
LD TR0
ANDNOT W58.07  ; #7位有电池
RSET H58.07  ; #7位有电池(记忆)
LD TR0
ANDNOT W58.08  ; #8位有电池
RSET H58.08  ; #8位有电池(记忆)
LD TR0
ANDNOT W58.09  ; #9位有电池
RSET H58.09  ; #9位有电池(记忆)
LD TR0
ANDNOT W58.10  ; #10位有电池
RSET H58.10  ; #10位有电池(记忆)
LD TR0
ANDNOT W58.11  ; #11位有电池
RSET H58.11  ; #11位有电池(记忆)
LD TR0
ANDNOT W58.12  ; #12位有电池
RSET H58.12  ; #12位有电池(记忆)

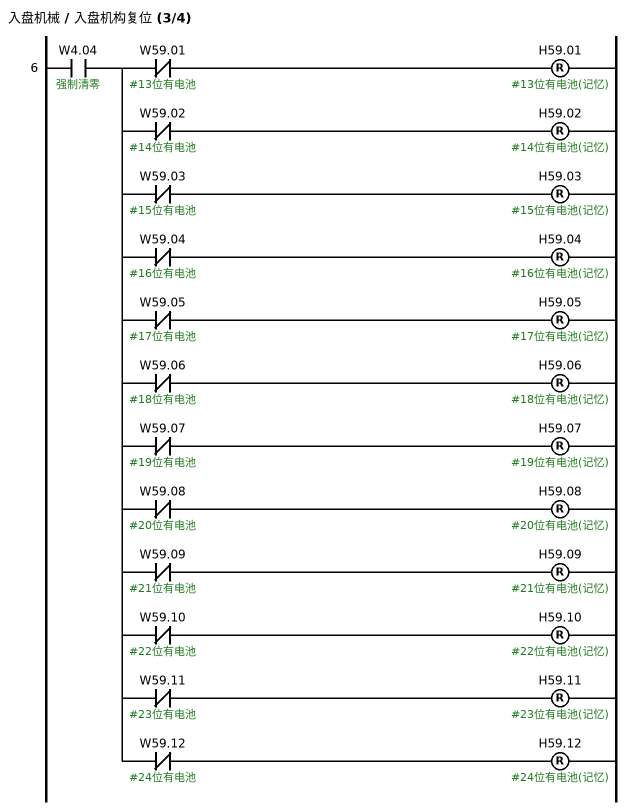
; rung 6
LD W4.04  ; 强制清零
OUT TR0
ANDNOT W59.01  ; #13位有电池
RSET H59.01  ; #13位有电池(记忆)
LD TR0
ANDNOT W59.02  ; #14位有电池
RSET H59.02  ; #14位有电池(记忆)
LD TR0
ANDNOT W59.03  ; #15位有电池
RSET H59.03  ; #15位有电池(记忆)
LD TR0
ANDNOT W59.04  ; #16位有电池
RSET H59.04  ; #16位有电池(记忆)
LD TR0
ANDNOT W59.05  ; #17位有电池
RSET H59.05  ; #17位有电池(记忆)
LD TR0
ANDNOT W59.06  ; #18位有电池
RSET H59.06  ; #18位有电池(记忆)
LD TR0
ANDNOT W59.07  ; #19位有电池
RSET H59.07  ; #19位有电池(记忆)
LD TR0
ANDNOT W59.08  ; #20位有电池
RSET H59.08  ; #20位有电池(记忆)
LD TR0
ANDNOT W59.09  ; #21位有电池
RSET H59.09  ; #21位有电池(记忆)
LD TR0
ANDNOT W59.10  ; #22位有电池
RSET H59.10  ; #22位有电池(记忆)
LD TR0
ANDNOT W59.11  ; #23位有电池
RSET H59.11  ; #23位有电池(记忆)
LD TR0
ANDNOT W59.12  ; #24位有电池
RSET H59.12  ; #24位有电池(记忆)

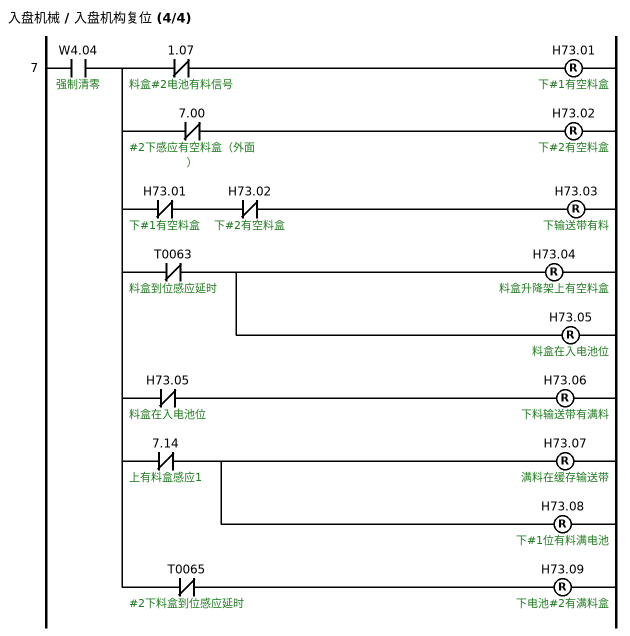
; rung 7
LD W4.04  ; 强制清零
OUT TR0
ANDNOT 1.07  ; 料盒#2电池有料信号
RSET H73.01  ; 下#1有空料盒
LD TR0
ANDNOT 7.00  ; #2下感应有空料盒（外面）
RSET H73.02  ; 下#2有空料盒
LD TR0
ANDNOT H73.01  ; 下#1有空料盒
ANDNOT H73.02  ; 下#2有空料盒
RSET H73.03  ; 下输送带有料
LD TR0
ANDNOT T0063  ; 料盒到位感应延时
RSET H73.04  ; 料盒升降架上有空料盒
RSET H73.05  ; 料盒在入电池位
LD TR0
ANDNOT H73.05  ; 料盒在入电池位
RSET H73.06  ; 下料输送带有满料
LD TR0
ANDNOT 7.14  ; 上有料盒感应1
RSET H73.07  ; 满料在缓存输送带
RSET H73.08  ; 下#1位有料满电池
LD TR0
ANDNOT T0065  ; #2下料盒到位感应延时
RSET H73.09  ; 下电池#2有满料盒

### Section END
; rung 0
END(001)